FUNCTION FC_GetMin3Lreals : LREAL		// Returns the minimum of specified values 
VAR_INPUT
	iLreal1:	LREAL;
	iLreal2:	LREAL;
	iLreal3:	LREAL;
END_VAR

FC_GetMin3Lreals := MIN(iLreal1, iLreal2);
FC_GetMin3Lreals := MIN(FC_GetMin3Lreals, iLreal3);

END_FUNCTION

(* stored: Version 1.1.0.1, ProductVersion 3.1.4026.18
   POU FC_GetMin3Lreals: Id {f17e01d6-e5bb-423a-bd3f-aaad92e206b4}, SpecialFunc None *)
